FUNCTION_BLOCK LWORD2LWORD
  {SET_ATTRIBUTE(OpcUa, SERVICE)}
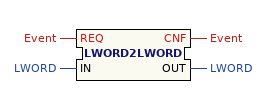
  EVENT_INPUT
    REQ;
  END_EVENT
  EVENT_OUTPUT
    CNF;
  END_EVENT
  VAR_INPUT
    IN : LWORD;
  END_VAR
  VAR_OUTPUT
    OUT : LWORD;
  END_VAR
END_FUNCTION_BLOCK
